// TIA Portal V17 export
// export: Created 2024-06-16T17:47:31.9789088Z, ExportSetting WithDefaults, DisplayName Totally Integrated Automation Portal, DisplayVersion V17, DisplayName TIA Portal Openness, DisplayVersion V17, DisplayName TIA Portal Version Control Interface, DisplayVersion V17, DisplayName STEP 7 Professional, DisplayVersion V17, DisplayName STEP 7 Safety, DisplayVersion V17, DisplayName WinCC Professional, DisplayVersion V17
DATA_BLOCK "G7A_St3_Init"   // DB310
VERSION : 0.1
// stored: AutoNumber false, DBAccessibleFromOPCUA true, DBAccessibleFromWebserver true, InstanceOfName G7A_St3_Init_FB, InstanceOfType FB
"G7A_St3_Init_FB"
   // VAR_OUTPUT
   //    "Step" : Int;
   // END_VAR
   // VAR
   //    Step_100 { ExternalAccessible := 'False'; ExternalVisible := 'False'; ExternalWritable := 'False'} : Int;
   //    Authorization : Bool;
   // END_VAR
BEGIN
END_DATA_BLOCK
